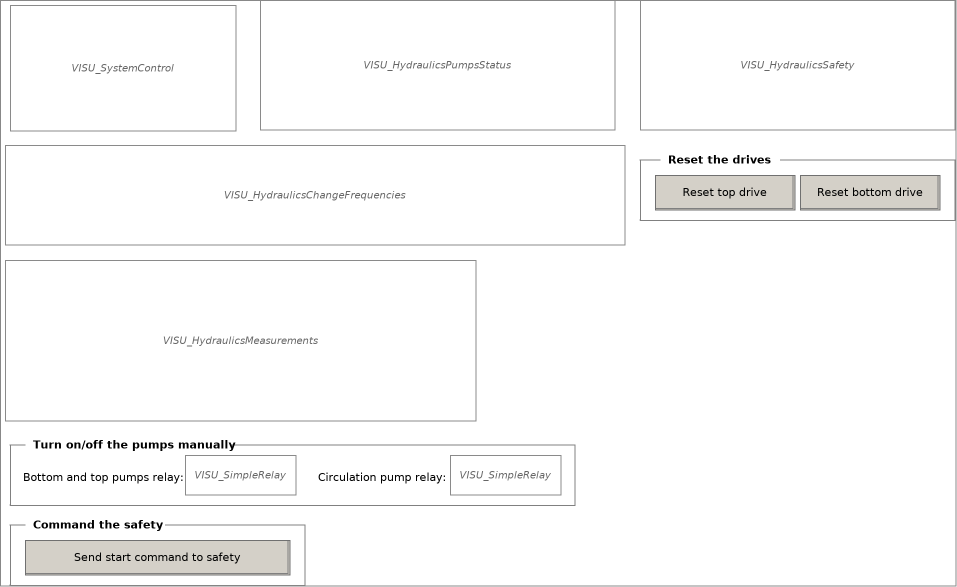
VISUALIZATION VISU_HydraulicsTechnical  // 957x587
VAR_IN_OUT
	ref : Hydraulics;
    widget : HydraulicsWidget;
    ref_safety : SafetyHydraulics;
END_VAR
    Polyline (25,445) (10,445) (10,505) (575,505) (575,445) (230,445)
    Frame (10,5 226x126)
        shows VISU_SystemControl(status := widget.actualStatus, button_initialize := widget.button_initialize, button_operating := widget.button_operating, button_locking := widget.button_locking)
    Frame (260,0 355x130)
        shows VISU_HydraulicsPumpsStatus(ref := ref, widget := widget, ref_safety := ref_safety)
    Frame (640,0 315x130)
        shows VISU_HydraulicsSafety(ref := ref, widget := widget, ref_safety := ref_safety)
    Frame (5,145 620x100)
        shows VISU_HydraulicsChangeFrequencies(ref := ref, widget := widget)
    Frame (5,260 471x161)
        shows VISU_HydraulicsMeasurements(ref := ref, widget := widget)
    Frame (185,455 111x40)
        shows VISU_SimpleRelay(ref := ref.parts.pumpsPowerRelay, widget := widget.pumpsPowerRelay)
    Label (20,460 165x35), "Bottom and top pumps relay:"
    Label (30,435 255x20), "Turn on/off the pumps manually"
    Polyline (25,525) (10,525) (10,585) (305,585) (305,525) (165,525)
    Label (30,515 135x20), "Command the safety"
    Button (25,540 265x35), "Send start command to safety", input disabled if: ref_safety.processes.startupPumps.statuses.enabledStatus.disabled
        OnMouseClick: execute { ref_safety.processes.startupPumps.do_request := TRUE; }
    Polyline (660,160) (640,160) (640,220) (955,220) (955,160) (780,160)
    Label (665,150 110x20), "Reset the drives"
    Button (655,175 140x35), "Reset top drive", input disabled if: ref.parts.top.processes.resetDrive.statuses.enabledStatus.disabled
        OnMouseClick: execute { ref.parts.top.processes.resetDrive.do_request := TRUE; }
    Button (800,175 140x35), "Reset bottom drive", input disabled if: ref.parts.bottom.processes.resetDrive.statuses.enabledStatus.disabled
        OnMouseClick: execute { ref.parts.bottom.processes.resetDrive.do_request := TRUE; }
    Label (315,460 145x35), "Circulation pump relay:"
    Frame (450,455 111x40)
        shows VISU_SimpleRelay(ref := ref.parts.circulationPumpRelay, widget := widget.circulationPumpRelay)
END_VISUALIZATION

(* stored: Version 1.1.0.1, ProductVersion 3.1.4019.2
   Visu VISU_HydraulicsTechnical: Id {3ed1b597-3dbd-4cf6-8116-68cd47401979} *)
